// SIMATIC S7-200 project (STEP 7-Micro/WIN), CPU 226 CN REL 02.01

ORGANIZATION_BLOCK 主程序:OB1
TITLE=程序注释
BEGIN
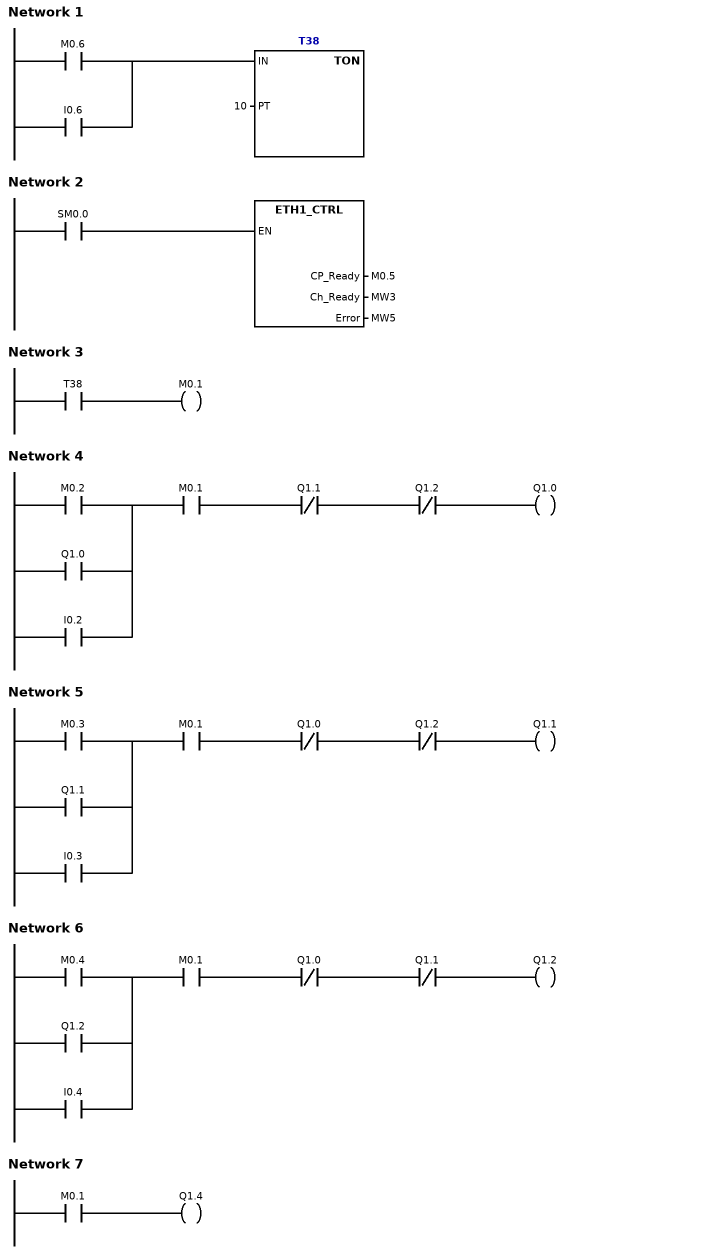
Network 1
LD     M0.6
O      I0.6
TON    T38, 10
Network 2
LD     SM0.0
CALL   ETH1_CTRL:SBR1, M0.5, MW3, MW5
Network 3
LD     T38
=      M0.1
Network 4
LD     M0.2
O      Q1.0
O      I0.2
A      M0.1
AN     Q1.1
AN     Q1.2
=      Q1.0
Network 5
LD     M0.3
O      Q1.1
O      I0.3
A      M0.1
AN     Q1.0
AN     Q1.2
=      Q1.1
Network 6
LD     M0.4
O      Q1.2
O      I0.4
A      M0.1
AN     Q1.0
AN     Q1.1
=      Q1.2
Network 7
LD     M0.1
=      Q1.4
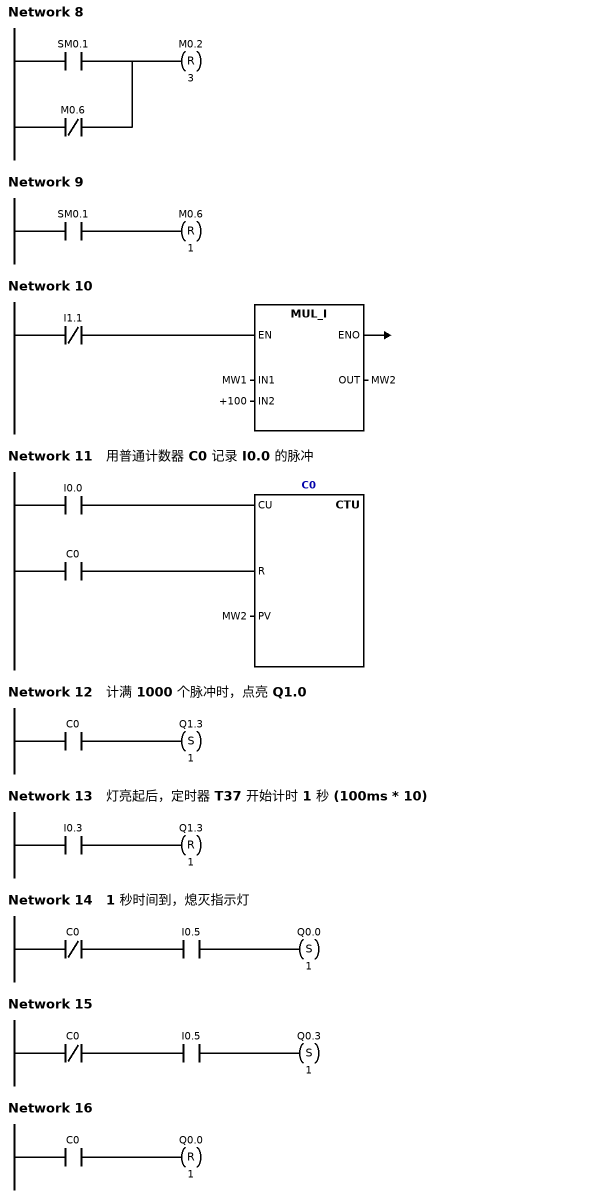
Network 8
LD     SM0.1
ON     M0.6
R      M0.2, 3
Network 9
LD     SM0.1
R      M0.6, 1
Network 10
LDN    I1.1
MOVW   MW1, MW2
*I     +100, MW2
Network 11 //  用普通计数器 C0 记录 I0.0 的脉冲
// 计数输入 (CU)：只读取 I0.0 (A相) 的脉冲
// 复位输入 (R)：当 C0 计满 1000 时，自己触发复位
// 预置值 (PV)：1000线编码器，设为1000就是一圈
LD     I0.0
LD     C0
CTU    C0, MW2
Network 12 //  计满 1000 个脉冲时，点亮 Q1.0
// 当 C0 到达 1000 的那个瞬间，C0位接通
// 置位 Q1.0（点亮指示灯）
LD     C0
S      Q1.3, 1
Network 13 //  灯亮起后，定时器 T37 开始计时 1 秒 (100ms * 10)
// 只要 Q1.0 亮着
// 启动 T37，延时 1 秒
LD     I0.3
R      Q1.3, 1
Network 14 //  1 秒时间到，熄灭指示灯
// 当延时到达 1 秒
// 复位 Q1.0（熄灭灯），同时 T37 也会自动复位
LDN    C0
A      I0.5
S      Q0.0, 1
Network 15
LDN    C0
A      I0.5
S      Q0.3, 1
Network 16
LD     C0
R      Q0.0, 1
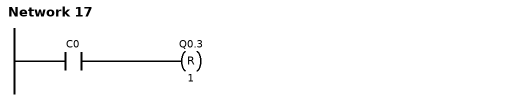
Network 17
LD     C0
R      Q0.3, 1
END_ORGANIZATION_BLOCK

// SBR1: protected block, not included

SUBROUTINE_BLOCK HSC_INIT:SBR2
TITLE=
BEGIN
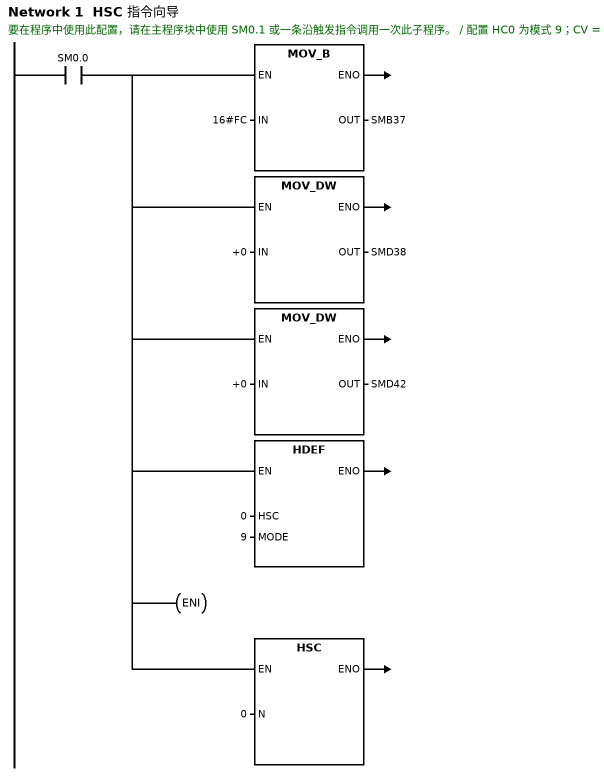
Network 1 // HSC 指令向导
// 要在程序中使用此配置，请在主程序块中使用 SM0.1 或一条沿触发指令调用一次此子程序。
// 配置 HC0 为模式 9；CV = 0； PV = 0；增计数；
// 开放中断和启动计数器。
// 
//设置控制位：增计数；1X 速率；已使能；
//装载 CV
//装载 PV
LD     SM0.0
MOVB   16#FC, SMB37
MOVD   +0, SMD38
MOVD   +0, SMD42
HDEF   0, 9
ENI
HSC    0
END_SUBROUTINE_BLOCK

// (further data pages could not be read)
